FUNCTION_BLOCK I_MSS (* Machine Selected Speed MSS *)
  (* Standard: ISO 11783-7; Classification: PGN 61474; Function: Machine Selected Speed MSS; Description: Copyright (c) 2024 HR Agrartechnik GmbH This program and the accompanying materials are made available under the terms of the Eclipse Public License 2.0 which is available at https://www.eclipse.org/legal/epl-2.0/ SPDX-License-Identifier: EPL-2.0 Message that provides the current machine selected speed, direction and source parameters. https://docs.ms-muc-docs.de/projects/isobus-other-docs/de/latest/PGN/PGN_61474.html *)
  (* Version 1.0, 2024-07-09, Franz Höpfinger, HR Agrartechnik GmbH *)
  PACKAGE isobus::tecu;
  (* Documentation:
  Machine Selected Speed MSS
   TIMEOUT / IND Vertrag: TIMEOUT feuert ausschliesslich beim tatsaechlichen Eintreten eines Timeouts (Q_timeout wird true). Das Zuruecksetzen von Q_timeout auf false (Timeout vorbei) wird bewusst NICHT nochmal separat ueber TIMEOUT gemeldet, sondern kommt ueber IND - das feuert bei jedem Zyklus ohne aktiven Timeout und publiziert Q_timeout mit. Nachgeschaltete Bausteine, die auf das Ende eines Timeouts reagieren muessen, werten dafuer IND mit Q_timeout==false aus, nicht ein zweites TIMEOUT-Event.
  *)
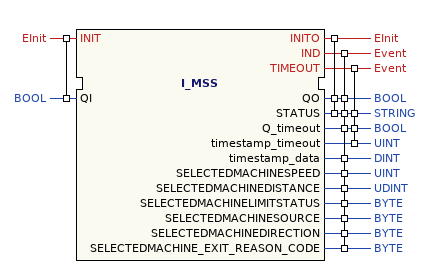
  EVENT_INPUT
    INIT : EInit WITH QI; (* Service Initialization *)
  END_EVENT
  EVENT_OUTPUT
    INITO : EInit WITH QO, STATUS; (* Initialization Confirm *)
    IND WITH QO, timestamp_data, STATUS, Q_timeout, SELECTEDMACHINESPEED, SELECTEDMACHINEDISTANCE, SELECTEDMACHINELIMITSTATUS, SELECTEDMACHINESOURCE, SELECTEDMACHINEDIRECTION, SELECTEDMACHINE_EXIT_REASON_CODE; (* Indication from Resource - feuert bei jedem Zyklus ohne aktiven Timeout und publiziert dabei auch den Reset von Q_timeout auf false. *)
    TIMEOUT WITH timestamp_timeout, STATUS, Q_timeout; (* Feuert ausschliesslich beim tatsaechlichen Eintreten eines Timeouts (Entry-Trigger). Das Zuruecksetzen von Q_timeout auf false wird NICHT hier, sondern ueber IND gemeldet. *)
  END_EVENT
  VAR_INPUT
    QI : BOOL; (* Event Input Qualifier *)
  END_VAR
  VAR_OUTPUT
    QO : BOOL; (* Event Output Qualifier *)
    STATUS : STRING;
    Q_timeout : BOOL;
    timestamp_timeout : UINT;
    timestamp_data : DINT;
    SELECTEDMACHINESPEED : UINT := UINT#16#FFFF; (* Machine selected speed (see Attributes for Details) *) {SET_ATTRIBUTE(SPN, 4305)} {SET_ATTRIBUTE(SP_Name, 'Machine selected speed')} {SET_ATTRIBUTE(SP_Position_In_PG, '1-2')} {SET_ATTRIBUTE(SP_Length, 16)} (* 16 bits *) {SET_ATTRIBUTE(Scaling, '0.001 m/s/bit, upper byte 0.256 m/s/bit')} {SET_ATTRIBUTE(Offset, )} {SET_ATTRIBUTE(Link, 'https://docs.ms-muc-docs.de/projects/isobus-other-docs/de/latest/PGN/PGN_61474.html#spn-4305-machine-selected-speed')}
    SELECTEDMACHINEDISTANCE : UDINT := UDINT#16#FFFFFFFF; (* Machine selected distance (see Attributes for Details) *) {SET_ATTRIBUTE(SPN, 4306)} {SET_ATTRIBUTE(SP_Name, 'Machine selected distance')} {SET_ATTRIBUTE(SP_Position_In_PG, '3-6')} {SET_ATTRIBUTE(SP_Length, 32)} (* 32 bits *) {SET_ATTRIBUTE(Scaling, '0.001 m/bit')} {SET_ATTRIBUTE(Offset, )} {SET_ATTRIBUTE(Link, 'https://docs.ms-muc-docs.de/projects/isobus-other-docs/de/latest/PGN/PGN_61474.html#spn-4306-machine-selected-distance')}
    SELECTEDMACHINELIMITSTATUS : BYTE := BYTE#16#FF; (* Machine selected speed limit status *) {SET_ATTRIBUTE(SPN, 4307)} {SET_ATTRIBUTE(SP_Name, 'Machine selected speed limit status')} {SET_ATTRIBUTE(SP_Position_In_PG, '8.6')} {SET_ATTRIBUTE(SP_Length, 3)} (* 3 bits *) {SET_ATTRIBUTE(Scaling, '8 states/3 bit')} {SET_ATTRIBUTE(Offset, )} {SET_ATTRIBUTE(Link, 'https://docs.ms-muc-docs.de/projects/isobus-other-docs/de/latest/PGN/PGN_61474.html#spn-4307-machine-selected-speed-limit-status')}
    SELECTEDMACHINESOURCE : BYTE := BYTE#16#FF; (* Machine selected speed source *) {SET_ATTRIBUTE(SPN, 4308)} {SET_ATTRIBUTE(SP_Name, 'Machine selected speed source')} {SET_ATTRIBUTE(SP_Position_In_PG, '8.3')} {SET_ATTRIBUTE(SP_Length, 3)} (* 3 bits *) {SET_ATTRIBUTE(Scaling, '8 states/3 bit')} {SET_ATTRIBUTE(Offset, )} {SET_ATTRIBUTE(Link, 'https://docs.ms-muc-docs.de/projects/isobus-other-docs/de/latest/PGN/PGN_61474.html#spn-4308-machine-selected-speed-source')}
    SELECTEDMACHINEDIRECTION : BYTE := BYTE#16#FF; (* Machine selected direction (see Attributes for Details) *) {SET_ATTRIBUTE(SPN, 4309)} {SET_ATTRIBUTE(SP_Name, 'Machine selected direction')} {SET_ATTRIBUTE(SP_Position_In_PG, '8.1')} {SET_ATTRIBUTE(SP_Length, 2)} (* 2 bits *) {SET_ATTRIBUTE(Scaling, '4 states/2 bit')} {SET_ATTRIBUTE(Offset, )} {SET_ATTRIBUTE(Link, 'https://docs.ms-muc-docs.de/projects/isobus-other-docs/de/latest/PGN/PGN_61474.html#spn-4309-machine-selected-direction')}
    SELECTEDMACHINE_EXIT_REASON_CODE : BYTE := BYTE#16#FF; (* Machine selected speed exit/reason code *) {SET_ATTRIBUTE(SPN, 5818)} {SET_ATTRIBUTE(SP_Name, 'Machine selected speed exit/reason code')} {SET_ATTRIBUTE(SP_Position_In_PG, '7.1')} {SET_ATTRIBUTE(SP_Length, 6)} (* 6 bits *) {SET_ATTRIBUTE(Scaling, '64 states/6 bit')} {SET_ATTRIBUTE(Offset, )} {SET_ATTRIBUTE(Link, 'https://docs.ms-muc-docs.de/projects/isobus-other-docs/de/latest/PGN/PGN_61474.html#spn-5818-machine-selected-speed-exit-reason-code')}
  END_VAR
END_FUNCTION_BLOCK
